{attribute 'qualified_only'}
{attribute 'strict'}
TYPE ComState :
(
	Idle, Send, Recv, Process, WaitForReceive, WaitForTransmit, WaitForInit, WaitForNotInit, ClearBuffer, RecvSetUp
);
END_TYPE

(* stored: Version 1.1.0.1, ProductVersion 3.1.4024.15
   DUT ComState: Id {6439d4cc-5dd1-49c3-9aab-80678a68b937} *)
